ABB RAPID module: Codigo Rappid

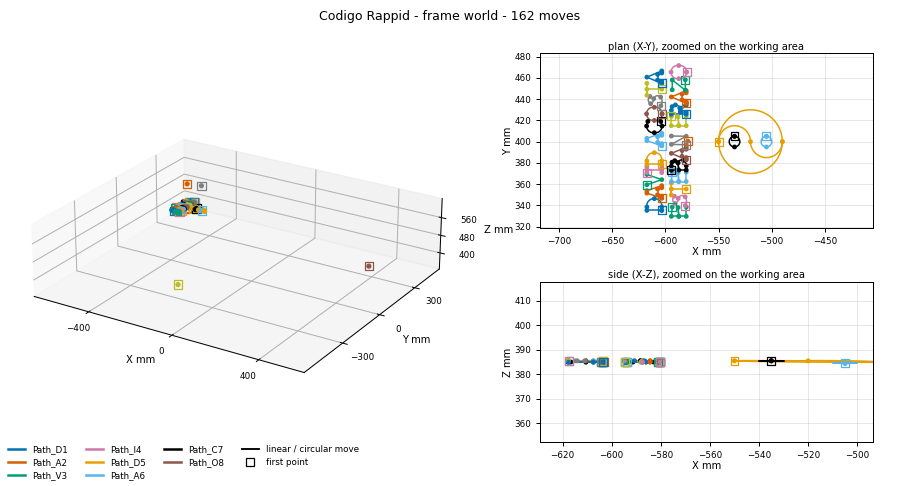
[picture p0: tool path of Codigo Rappid in frame world, 162 of 163 moves have a stored position in this frame; points joined in program order, loops and branches not executed]
MODULE Module1
    PERS tooldata Porta_Marcador:=[TRUE,[[111.723,0,111.723],[0.923879533,0,0.382683432,0]],[1,[0,0,1],[1,0,0,0],0,0,0]];
    TASK PERS wobjdata Workobject_2:=[FALSE,TRUE,"",[[-160,-80,65],[1,0,0,0]],[[-480,560,320],[0,1,0,0]]];
    CONST robtarget Target_10:=[[36.486,144.721,0],[1,0,0,0],[0,0,0,0],[9E+09,9E+09,9E+09,9E+09,9E+09,9E+09]];
    CONST robtarget Target_20:=[[22.486,144.721,-0.5],[1,0,0,0],[0,0,0,0],[9E+09,9E+09,9E+09,9E+09,9E+09,9E+09]];
    CONST robtarget Target_30:=[[22.486,141.533,-0.5],[1,0,0,0],[0,0,0,0],[9E+09,9E+09,9E+09,9E+09,9E+09,9E+09]];
    CONST robtarget Target_40:=[[23.598,136.519,-0.5],[1,0,0,0],[0,0,0,0],[9E+09,9E+09,9E+09,9E+09,9E+09,9E+09]];
    CONST robtarget Target_50:=[[29.498,133.682,0],[1,0,0,0],[0,0,0,0],[9E+09,9E+09,9E+09,9E+09,9E+09,9E+09]];
    CONST robtarget Target_60:=[[35.363,136.541,-0.5],[1,0,0,0],[0,0,0,0],[9E+09,9E+09,9E+09,9E+09,9E+09,9E+09]];
    CONST robtarget Target_70:=[[36.486,141.499,0],[1,0,0,0],[0,0,0,0],[9E+09,9E+09,9E+09,9E+09,9E+09,9E+09]];
    CONST robtarget Target_80:=[[36.486,133.172,-0.5],[1,0,0,0],[0,0,0,0],[9E+09,9E+09,9E+09,9E+09,9E+09,9E+09]];
    CONST robtarget Target_90:=[[22.486,128.452,-0.5],[1,0,0,0],[0,0,0,0],[9E+09,9E+09,9E+09,9E+09,9E+09,9E+09]];
    CONST robtarget Target_100:=[[22.486,126.161,0],[1,0,0,0],[0,0,0,0],[9E+09,9E+09,9E+09,9E+09,9E+09,9E+09]];
    CONST robtarget Target_110:=[[36.486,121.441,-0.5],[1,0,0,0],[0,0,0,0],[9E+09,9E+09,9E+09,9E+09,9E+09,9E+09]];
    CONST robtarget Target_120:=[[36.486,123.404,0],[1,0,0,0],[0,0,0,0],[9E+09,9E+09,9E+09,9E+09,9E+09,9E+09]];
    CONST robtarget Target_130:=[[32.572,124.674,-0.5],[1,0,0,0],[0,0,0,0],[9E+09,9E+09,9E+09,9E+09,9E+09,9E+09]];
    CONST robtarget Target_140:=[[32.572,130.018,0],[1,0,0,0],[0,0,0,0],[9E+09,9E+09,9E+09,9E+09,9E+09,9E+09]];
    CONST robtarget Target_150:=[[36.486,131.289,-0.5],[1,0,0,0],[0,0,0,0],[9E+09,9E+09,9E+09,9E+09,9E+09,9E+09]];
    CONST robtarget Target_160:=[[22.486,120.613,-0.5],[1,0,0,0],[0,0,0,0],[9E+09,9E+09,9E+09,9E+09,9E+09,9E+09]];
    CONST robtarget Target_170:=[[36.486,115.785,-0.5],[1,0,0,0],[0,0,0,0],[9E+09,9E+09,9E+09,9E+09,9E+09,9E+09]];
    CONST robtarget Target_180:=[[22.486,110.907,-0.5],[1,0,0,0],[0,0,0,0],[9E+09,9E+09,9E+09,9E+09,9E+09,9E+09]];
    CONST robtarget Target_190:=[[22.486,109.165,-0.5],[1,0,0,0],[0,0,0,0],[9E+09,9E+09,9E+09,9E+09,9E+09,9E+09]];
    CONST robtarget Target_200:=[[22.486,103.742,-0.5],[1,0,0,0],[0,0,0,0],[9E+09,9E+09,9E+09,9E+09,9E+09,9E+09]];
    CONST robtarget Target_210:=[[22.486,106.454,-0.5],[1,0,0,0],[0,0,0,0],[9E+09,9E+09,9E+09,9E+09,9E+09,9E+09]];
    CONST robtarget Target_220:=[[36.486,106.454,-0.25],[1,0,0,0],[0,0,0,0],[9E+09,9E+09,9E+09,9E+09,9E+09,9E+09]];
    CONST robtarget Target_230:=[[36.486,109.165,-0.25],[1,0,0,0],[0,0,0,0],[9E+09,9E+09,9E+09,9E+09,9E+09,9E+09]];
    CONST robtarget Target_240:=[[36.486,103.742,0],[1,0,0,0],[0,0,0,0],[9E+09,9E+09,9E+09,9E+09,9E+09,9E+09]];
    CONST robtarget Target_250:=[[36.486,101.439,0],[1,0,0,0],[0,0,0,0],[9E+09,9E+09,9E+09,9E+09,9E+09,9E+09]];
    CONST robtarget Target_260:=[[22.486,101.439,-0.5],[1,0,0,0],[0,0,0,0],[9E+09,9E+09,9E+09,9E+09,9E+09,9E+09]];
    CONST robtarget Target_270:=[[22.486,98.251,-0.5],[1,0,0,0],[0,0,0,0],[9E+09,9E+09,9E+09,9E+09,9E+09,9E+09]];
    CONST robtarget Target_280:=[[23.598,93.237,-0.5],[1,0,0,0],[0,0,0,0],[9E+09,9E+09,9E+09,9E+09,9E+09,9E+09]];
    CONST robtarget Target_290:=[[29.498,90.4,0],[1,0,0,0],[0,0,0,0],[9E+09,9E+09,9E+09,9E+09,9E+09,9E+09]];
    CONST robtarget Target_300:=[[35.363,93.259,0],[1,0,0,0],[0,0,0,0],[9E+09,9E+09,9E+09,9E+09,9E+09,9E+09]];
    CONST robtarget Target_310:=[[36.486,98.217,0],[1,0,0,0],[0,0,0,0],[9E+09,9E+09,9E+09,9E+09,9E+09,9E+09]];
    CONST robtarget Target_320:=[[36.486,83.877,0],[1,0,0,0],[0,0,0,0],[9E+09,9E+09,9E+09,9E+09,9E+09,9E+09]];
    CONST robtarget Target_330:=[[22.486,79.157,-0.5],[1,0,0,0],[0,0,0,0],[9E+09,9E+09,9E+09,9E+09,9E+09,9E+09]];
    CONST robtarget Target_340:=[[22.486,76.866,-0.5],[1,0,0,0],[0,0,0,0],[9E+09,9E+09,9E+09,9E+09,9E+09,9E+09]];
    CONST robtarget Target_350:=[[36.486,72.146,0],[1,0,0,0],[0,0,0,0],[9E+09,9E+09,9E+09,9E+09,9E+09,9E+09]];
    CONST robtarget Target_360:=[[36.486,74.109,0],[1,0,0,0],[0,0,0,0],[9E+09,9E+09,9E+09,9E+09,9E+09,9E+09]];
    CONST robtarget Target_370:=[[32.572,75.379,-0.5],[1,0,0,0],[0,0,0,0],[9E+09,9E+09,9E+09,9E+09,9E+09,9E+09]];
    CONST robtarget Target_380:=[[32.572,80.723,0],[1,0,0,0],[0,0,0,0],[9E+09,9E+09,9E+09,9E+09,9E+09,9E+09]];
    CONST robtarget Target_390:=[[36.486,81.994,0],[1,0,0,0],[0,0,0,0],[9E+09,9E+09,9E+09,9E+09,9E+09,9E+09]];
    CONST robtarget Target_400:=[[35.533,60.994,0],[1,0,0,0],[0,0,0,0],[9E+09,9E+09,9E+09,9E+09,9E+09,9E+09]];
    CONST robtarget Target_410:=[[36.328,62.854,0],[1,0,0,0],[0,0,0,0],[9E+09,9E+09,9E+09,9E+09,9E+09,9E+09]];
    CONST robtarget Target_420:=[[36.736,65.35,0],[1,0,0,0],[0,0,0,0],[9E+09,9E+09,9E+09,9E+09,9E+09,9E+09]];
    CONST robtarget Target_430:=[[34.898,69.854,0],[1,0,0,0],[0,0,0,0],[9E+09,9E+09,9E+09,9E+09,9E+09,9E+09]];
    CONST robtarget Target_440:=[[29.498,71.613,0],[1,0,0,0],[0,0,0,0],[9E+09,9E+09,9E+09,9E+09,9E+09,9E+09]];
    CONST robtarget Target_450:=[[24.165,69.866,-0.5],[1,0,0,0],[0,0,0,0],[9E+09,9E+09,9E+09,9E+09,9E+09,9E+09]];
    CONST robtarget Target_460:=[[22.237,65.316,0],[1,0,0,0],[0,0,0,0],[9E+09,9E+09,9E+09,9E+09,9E+09,9E+09]];
    CONST robtarget Target_470:=[[22.6,62.854,0],[1,0,0,0],[0,0,0,0],[9E+09,9E+09,9E+09,9E+09,9E+09,9E+09]];
    CONST robtarget Target_480:=[[23.417,60.994,0],[1,0,0,0],[0,0,0,0],[9E+09,9E+09,9E+09,9E+09,9E+09,9E+09]];
    CONST robtarget Target_490:=[[36.781,53.869,0],[1,0,0,0],[0,0,0,0],[9E+09,9E+09,9E+09,9E+09,9E+09,9E+09]];
    CONST robtarget Target_500:=[[34.875,58.384,0],[1,0,0,0],[0,0,0,0],[9E+09,9E+09,9E+09,9E+09,9E+09,9E+09]];
    CONST robtarget Target_510:=[[29.486,60.052,-0.5],[1,0,0,0],[0,0,0,0],[9E+09,9E+09,9E+09,9E+09,9E+09,9E+09]];
    CONST robtarget Target_520:=[[24.086,58.373,-0.5],[1,0,0,0],[0,0,0,0],[9E+09,9E+09,9E+09,9E+09,9E+09,9E+09]];
    CONST robtarget Target_530:=[[22.191,53.869,-0.5],[1,0,0,0],[0,0,0,0],[9E+09,9E+09,9E+09,9E+09,9E+09,9E+09]];
    CONST robtarget Target_540:=[[24.086,49.353,-0.5],[1,0,0,0],[0,0,0,0],[9E+09,9E+09,9E+09,9E+09,9E+09,9E+09]];
    CONST robtarget Target_550:=[[29.486,47.674,-0.5],[1,0,0,0],[0,0,0,0],[9E+09,9E+09,9E+09,9E+09,9E+09,9E+09]];
    CONST robtarget Target_560:=[[34.875,49.353,-0.5],[1,0,0,0],[0,0,0,0],[9E+09,9E+09,9E+09,9E+09,9E+09,9E+09]];
    CONST robtarget Target_570:=[[35.647,46.324,0],[1,0,0,0],[0,0,0,0],[9E+09,9E+09,9E+09,9E+09,9E+09,9E+09]];
    CONST robtarget Target_580:=[[36.736,41.729,0],[1,0,0,0],[0,0,0,0],[9E+09,9E+09,9E+09,9E+09,9E+09,9E+09]];
    CONST robtarget Target_590:=[[35.465,38.076,0],[1,0,0,0],[0,0,0,0],[9E+09,9E+09,9E+09,9E+09,9E+09,9E+09]];
    CONST robtarget Target_600:=[[32.493,36.806,0],[1,0,0,0],[0,0,0,0],[9E+09,9E+09,9E+09,9E+09,9E+09,9E+09]];
    CONST robtarget Target_610:=[[28.964,39.585,-0.5],[1,0,0,0],[0,0,0,0],[9E+09,9E+09,9E+09,9E+09,9E+09,9E+09]];
    CONST robtarget Target_620:=[[28.227,42.456,-0.5],[1,0,0,0],[0,0,0,0],[9E+09,9E+09,9E+09,9E+09,9E+09,9E+09]];
    CONST robtarget Target_630:=[[26.049,44.282,-0.5],[1,0,0,0],[0,0,0,0],[9E+09,9E+09,9E+09,9E+09,9E+09,9E+09]];
    CONST robtarget Target_640:=[[23.848,41.389,-0.5],[1,0,0,0],[0,0,0,0],[9E+09,9E+09,9E+09,9E+09,9E+09,9E+09]];
    CONST robtarget Target_650:=[[25.368,37.486,-0.5],[1,0,0,0],[0,0,0,0],[9E+09,9E+09,9E+09,9E+09,9E+09,9E+09]];
    CONST robtarget Target_660:=[[36.486,30.713,-0.5],[1,0,0,0],[0,0,0,0],[9E+09,9E+09,9E+09,9E+09,9E+09,9E+09]];
    CONST robtarget Target_670:=[[22.486,30.713,-0.5],[1,0,0,0],[0,0,0,0],[9E+09,9E+09,9E+09,9E+09,9E+09,9E+09]];
    CONST robtarget Target_680:=[[22.486,36.34,-0.5],[1,0,0,0],[0,0,0,0],[9E+09,9E+09,9E+09,9E+09,9E+09,9E+09]];
    CONST robtarget Target_690:=[[22.486,25.086,-0.5],[1,0,0,0],[0,0,0,0],[9E+09,9E+09,9E+09,9E+09,9E+09,9E+09]];
    CONST robtarget Target_770:=[[36.486,25.177,0],[1,0,0,0],[0,0,0,0],[9E+09,9E+09,9E+09,9E+09,9E+09,9E+09]];
    CONST robtarget Target_780:=[[22.486,19.311,0],[1,0,0,0],[0,0,0,0],[9E+09,9E+09,9E+09,9E+09,9E+09,9E+09]];
    CONST robtarget Target_790:=[[36.486,13.446,0],[1,0,0,0],[0,0,0,0],[9E+09,9E+09,9E+09,9E+09,9E+09,9E+09]];
    CONST robtarget Target_800:=[[36.486,15.409,0],[1,0,0,0],[0,0,0,0],[9E+09,9E+09,9E+09,9E+09,9E+09,9E+09]];
    CONST robtarget Target_810:=[[32.572,16.679,0],[1,0,0,0],[0,0,0,0],[9E+09,9E+09,9E+09,9E+09,9E+09,9E+09]];
    CONST robtarget Target_820:=[[32.572,22.023,0],[1,0,0,0],[0,0,0,0],[9E+09,9E+09,9E+09,9E+09,9E+09,9E+09]];
    CONST robtarget Target_830:=[[36.486,23.293,0],[1,0,0,0],[0,0,0,0],[9E+09,9E+09,9E+09,9E+09,9E+09,9E+09]];
    CONST robtarget Target_Pastel_inicio:=[[61.043181897,79.487763711,-109.905526816],[0.928113719,0.029025657,-0.074070087,0.363697757],[1,-1,0,0],[9E+09,9E+09,9E+09,9E+09,9E+09,9E+09]];
    CONST robtarget Target_840:=[[46.365,141.579,0],[1,0,0,0],[0,0,0,0],[9E+09,9E+09,9E+09,9E+09,9E+09,9E+09]];
    CONST robtarget Target_850:=[[45.537,150.337,0],[1,0,0,0],[0,0,0,0],[9E+09,9E+09,9E+09,9E+09,9E+09,9E+09]];
    CONST robtarget Target_860:=[[52.537,150.337,0],[1,0,0,0],[0,0,0,0],[9E+09,9E+09,9E+09,9E+09,9E+09,9E+09]];
    CONST robtarget Target_870:=[[51.856,142.044,0],[1,0,0,0],[0,0,0,0],[9E+09,9E+09,9E+09,9E+09,9E+09,9E+09]];
    CONST robtarget Target_880:=[[59.537,150.337,0],[1,0,0,0],[0,0,0,0],[9E+09,9E+09,9E+09,9E+09,9E+09,9E+09]];
    CONST robtarget Target_890:=[[59.537,141.579,0],[1,0,0,0],[0,0,0,0],[9E+09,9E+09,9E+09,9E+09,9E+09,9E+09]];
    CONST robtarget Target_900:=[[58.697,140.229,0],[1,0,0,0],[0,0,0,0],[9E+09,9E+09,9E+09,9E+09,9E+09,9E+09]];
    CONST robtarget Target_910:=[[59.787,135.634,0],[1,0,0,0],[0,0,0,0],[9E+09,9E+09,9E+09,9E+09,9E+09,9E+09]];
    CONST robtarget Target_920:=[[58.516,131.981,0],[1,0,0,0],[0,0,0,0],[9E+09,9E+09,9E+09,9E+09,9E+09,9E+09]];
    CONST robtarget Target_930:=[[55.543,130.71,0],[1,0,0,0],[0,0,0,0],[9E+09,9E+09,9E+09,9E+09,9E+09,9E+09]];
    CONST robtarget Target_940:=[[52.015,133.49,-0.5],[1,0,0,0],[0,0,0,0],[9E+09,9E+09,9E+09,9E+09,9E+09,9E+09]];
    CONST robtarget Target_950:=[[51.278,136.36,-0.5],[1,0,0,0],[0,0,0,0],[9E+09,9E+09,9E+09,9E+09,9E+09,9E+09]];
    CONST robtarget Target_960:=[[49.099,138.186,-0.5],[1,0,0,0],[0,0,0,0],[9E+09,9E+09,9E+09,9E+09,9E+09,9E+09]];
    CONST robtarget Target_970:=[[46.898,135.293,0],[1,0,0,0],[0,0,0,0],[9E+09,9E+09,9E+09,9E+09,9E+09,9E+09]];
    CONST robtarget Target_980:=[[48.419,131.391,0],[1,0,0,0],[0,0,0,0],[9E+09,9E+09,9E+09,9E+09,9E+09,9E+09]];
    CONST robtarget Target_990:=[[59.537,124.618,0],[1,0,0,0],[0,0,0,0],[9E+09,9E+09,9E+09,9E+09,9E+09,9E+09]];
    CONST robtarget Target_1000:=[[45.537,124.618,-0.5],[1,0,0,0],[0,0,0,0],[9E+09,9E+09,9E+09,9E+09,9E+09,9E+09]];
    CONST robtarget Target_1010:=[[45.537,130.245,-0.5],[1,0,0,0],[0,0,0,0],[9E+09,9E+09,9E+09,9E+09,9E+09,9E+09]];
    CONST robtarget Target_1020:=[[45.537,118.99,0],[1,0,0,0],[0,0,0,0],[9E+09,9E+09,9E+09,9E+09,9E+09,9E+09]];
    CONST robtarget Target_1030:=[[46.365,108.814,0],[1,0,0,0],[0,0,0,0],[9E+09,9E+09,9E+09,9E+09,9E+09,9E+09]];
    CONST robtarget Target_1040:=[[45.537,117.572,-0.5],[1,0,0,0],[0,0,0,0],[9E+09,9E+09,9E+09,9E+09,9E+09,9E+09]];
    CONST robtarget Target_1050:=[[52.537,117.572,-0.5],[1,0,0,0],[0,0,0,0],[9E+09,9E+09,9E+09,9E+09,9E+09,9E+09]];
    CONST robtarget Target_1060:=[[51.856,109.279,-0.5],[1,0,0,0],[0,0,0,0],[9E+09,9E+09,9E+09,9E+09,9E+09,9E+09]];
    CONST robtarget Target_1070:=[[59.537,117.572,-0.5],[1,0,0,0],[0,0,0,0],[9E+09,9E+09,9E+09,9E+09,9E+09,9E+09]];
    CONST robtarget Target_1080:=[[59.537,108.814,0],[1,0,0,0],[0,0,0,0],[9E+09,9E+09,9E+09,9E+09,9E+09,9E+09]];
    CONST robtarget Target_1090:=[[45.537,106.772,0],[1,0,0,0],[0,0,0,0],[9E+09,9E+09,9E+09,9E+09,9E+09,9E+09]];
    CONST robtarget Target_1100:=[[59.537,106.772,0],[1,0,0,0],[0,0,0,0],[9E+09,9E+09,9E+09,9E+09,9E+09,9E+09]];
    CONST robtarget Target_1110:=[[59.537,102.755,0],[1,0,0,0],[0,0,0,0],[9E+09,9E+09,9E+09,9E+09,9E+09,9E+09]];
    CONST robtarget Target_1120:=[[59.276,100.424,0],[1,0,0,0],[0,0,0,0],[9E+09,9E+09,9E+09,9E+09,9E+09,9E+09]];
    CONST robtarget Target_1130:=[[57.081,97.673,0],[1,0,0,0],[0,0,0,0],[9E+09,9E+09,9E+09,9E+09,9E+09,9E+09]];
    CONST robtarget Target_1140:=[[52.996,97.962,0],[1,0,0,0],[0,0,0,0],[9E+09,9E+09,9E+09,9E+09,9E+09,9E+09]];
    CONST robtarget Target_1150:=[[51.754,99.896,-0.5],[1,0,0,0],[0,0,0,0],[9E+09,9E+09,9E+09,9E+09,9E+09,9E+09]];
    CONST robtarget Target_1160:=[[52.537,106.772,-0.5],[1,0,0,0],[0,0,0,0],[9E+09,9E+09,9E+09,9E+09,9E+09,9E+09]];
    CONST robtarget Target_1170:=[[50.461,98.456,0],[1,0,0,0],[0,0,0,0],[9E+09,9E+09,9E+09,9E+09,9E+09,9E+09]];
    CONST robtarget Target_1180:=[[48.691,97.934,0],[1,0,0,0],[0,0,0,0],[9E+09,9E+09,9E+09,9E+09,9E+09,9E+09]];
    CONST robtarget Target_1190:=[[47.154,98.28,0],[1,0,0,0],[0,0,0,0],[9E+09,9E+09,9E+09,9E+09,9E+09,9E+09]];
    CONST robtarget Target_1200:=[[46.104,99.386,0],[1,0,0,0],[0,0,0,0],[9E+09,9E+09,9E+09,9E+09,9E+09,9E+09]];
    CONST robtarget Target_1210:=[[45.537,103.062,-0.5],[1,0,0,0],[0,0,0,0],[9E+09,9E+09,9E+09,9E+09,9E+09,9E+09]];
    CONST robtarget Target_1220:=[[59.537,96.935,0],[1,0,0,0],[0,0,0,0],[9E+09,9E+09,9E+09,9E+09,9E+09,9E+09]];
    CONST robtarget Target_1230:=[[45.537,91.07,-0.5],[1,0,0,0],[0,0,0,0],[9E+09,9E+09,9E+09,9E+09,9E+09,9E+09]];
    CONST robtarget Target_1240:=[[59.537,85.204,0],[1,0,0,0],[0,0,0,0],[9E+09,9E+09,9E+09,9E+09,9E+09,9E+09]];
    CONST robtarget Target_1250:=[[59.537,87.167,0],[1,0,0,0],[0,0,0,0],[9E+09,9E+09,9E+09,9E+09,9E+09,9E+09]];
    CONST robtarget Target_1260:=[[55.623,88.438,-0.5],[1,0,0,0],[0,0,0,0],[9E+09,9E+09,9E+09,9E+09,9E+09,9E+09]];
    CONST robtarget Target_1270:=[[55.623,93.781,0],[1,0,0,0],[0,0,0,0],[9E+09,9E+09,9E+09,9E+09,9E+09,9E+09]];
    CONST robtarget Target_1280:=[[59.537,95.052,0],[1,0,0,0],[0,0,0,0],[9E+09,9E+09,9E+09,9E+09,9E+09,9E+09]];
    CONST robtarget Target_1290:=[[59.537,83.009,0],[1,0,0,0],[0,0,0,0],[9E+09,9E+09,9E+09,9E+09,9E+09,9E+09]];
    CONST robtarget Target_1300:=[[45.537,82.555,-0.5],[1,0,0,0],[0,0,0,0],[9E+09,9E+09,9E+09,9E+09,9E+09,9E+09]];
    CONST robtarget Target_1310:=[[59.537,74.903,0],[1,0,0,0],[0,0,0,0],[9E+09,9E+09,9E+09,9E+09,9E+09,9E+09]];
    CONST robtarget Target_1320:=[[45.537,74.727,-0.5],[1,0,0,0],[0,0,0,0],[9E+09,9E+09,9E+09,9E+09,9E+09,9E+09]];
    CONST robtarget Target_1340:=[[45.537,56.251,0],[1,0,0,0],[0,0,0,0],[9E+09,9E+09,9E+09,9E+09,9E+09,9E+09]];
    CONST robtarget Target_1350:=[[45.537,65.01,-0.5],[1,0,0,0],[0,0,0,0],[9E+09,9E+09,9E+09,9E+09,9E+09,9E+09]];
    CONST robtarget Target_1360:=[[52.537,65.01,-0.5],[1,0,0,0],[0,0,0,0],[9E+09,9E+09,9E+09,9E+09,9E+09,9E+09]];
    CONST robtarget Target_1370:=[[51.856,56.716,0],[1,0,0,0],[0,0,0,0],[9E+09,9E+09,9E+09,9E+09,9E+09,9E+09]];
    CONST robtarget Target_1380:=[[59.537,65.01,0],[1,0,0,0],[0,0,0,0],[9E+09,9E+09,9E+09,9E+09,9E+09,9E+09]];
    CONST robtarget Target_1390:=[[59.537,56.251,0],[1,0,0,0],[0,0,0,0],[9E+09,9E+09,9E+09,9E+09,9E+09,9E+09]];
    CONST robtarget Target_1400:=[[59.537,54.209,0],[1,0,0,0],[0,0,0,0],[9E+09,9E+09,9E+09,9E+09,9E+09,9E+09]];
    CONST robtarget Target_1410:=[[45.537,54.209,0],[1,0,0,0],[0,0,0,0],[9E+09,9E+09,9E+09,9E+09,9E+09,9E+09]];
    CONST robtarget Target_1420:=[[45.537,50.601,-0.5],[1,0,0,0],[0,0,0,0],[9E+09,9E+09,9E+09,9E+09,9E+09,9E+09]];
    CONST robtarget Target_1430:=[[45.667,48.588,-0.5],[1,0,0,0],[0,0,0,0],[9E+09,9E+09,9E+09,9E+09,9E+09,9E+09]];
    CONST robtarget Target_1440:=[[46.274,47.039,-0.5],[1,0,0,0],[0,0,0,0],[9E+09,9E+09,9E+09,9E+09,9E+09,9E+09]];
    CONST robtarget Target_1450:=[[47.494,45.876,-0.5],[1,0,0,0],[0,0,0,0],[9E+09,9E+09,9E+09,9E+09,9E+09,9E+09]];
    CONST robtarget Target_1460:=[[49.338,45.451,-0.5],[1,0,0,0],[0,0,0,0],[9E+09,9E+09,9E+09,9E+09,9E+09,9E+09]];
    CONST robtarget Target_1470:=[[51.907,46.233,-0.5],[1,0,0,0],[0,0,0,0],[9E+09,9E+09,9E+09,9E+09,9E+09,9E+09]];
    CONST robtarget Target_1480:=[[53.445,48.355,-0.5],[1,0,0,0],[0,0,0,0],[9E+09,9E+09,9E+09,9E+09,9E+09,9E+09]];
    CONST robtarget Target_1490:=[[59.537,43.84,0],[1,0,0,0],[0,0,0,0],[9E+09,9E+09,9E+09,9E+09,9E+09,9E+09]];
    CONST robtarget Target_1500:=[[59.537,45.791,0],[1,0,0,0],[0,0,0,0],[9E+09,9E+09,9E+09,9E+09,9E+09,9E+09]];
    CONST robtarget Target_1510:=[[53.966,50.216,0],[1,0,0,0],[0,0,0,0],[9E+09,9E+09,9E+09,9E+09,9E+09,9E+09]];
    CONST robtarget Target_1520:=[[53.966,52.349,0],[1,0,0,0],[0,0,0,0],[9E+09,9E+09,9E+09,9E+09,9E+09,9E+09]];
    CONST robtarget Target_1530:=[[59.537,52.349,0],[1,0,0,0],[0,0,0,0],[9E+09,9E+09,9E+09,9E+09,9E+09,9E+09]];
    CONST robtarget Target_1540:=[[59.537,43.84,0],[1,0,0,0],[0,0,0,0],[9E+09,9E+09,9E+09,9E+09,9E+09,9E+09]];
    CONST robtarget Target_1550:=[[45.537,37.906,-0.5],[1,0,0,0],[0,0,0,0],[9E+09,9E+09,9E+09,9E+09,9E+09,9E+09]];
    CONST robtarget Target_1560:=[[59.537,32.041,0],[1,0,0,0],[0,0,0,0],[9E+09,9E+09,9E+09,9E+09,9E+09,9E+09]];
    CONST robtarget Target_1570:=[[59.537,34.003,-0.25],[1,0,0,0],[0,0,0,0],[9E+09,9E+09,9E+09,9E+09,9E+09,9E+09]];
    CONST robtarget Target_1580:=[[55.623,35.274,-0.5],[1,0,0,0],[0,0,0,0],[9E+09,9E+09,9E+09,9E+09,9E+09,9E+09]];
    CONST robtarget Target_1590:=[[55.623,40.618,0],[1,0,0,0],[0,0,0,0],[9E+09,9E+09,9E+09,9E+09,9E+09,9E+09]];
    CONST robtarget Target_1600:=[[59.537,41.888,-0.25],[1,0,0,0],[0,0,0,0],[9E+09,9E+09,9E+09,9E+09,9E+09,9E+09]];
    CONST robtarget Target_1610:=[[58.709,21.785,0],[1,0,0,0],[0,0,0,0],[9E+09,9E+09,9E+09,9E+09,9E+09,9E+09]];
    CONST robtarget Target_1620:=[[58.669,31.564,-0.5],[1,0,0,0],[0,0,0,0],[9E+09,9E+09,9E+09,9E+09,9E+09,9E+09]];
    CONST robtarget Target_1630:=[[46.377,21.977,0],[1,0,0,0],[0,0,0,0],[9E+09,9E+09,9E+09,9E+09,9E+09,9E+09]];
    CONST robtarget Target_1640:=[[46.365,31.224,-0.5],[1,0,0,0],[0,0,0,0],[9E+09,9E+09,9E+09,9E+09,9E+09,9E+09]];
    CONST robtarget Target_1650:=[[59.832,14.558,0],[1,0,0,0],[0,0,0,0],[9E+09,9E+09,9E+09,9E+09,9E+09,9E+09]];
    CONST robtarget Target_1660:=[[57.926,19.073,0],[1,0,0,0],[0,0,0,0],[9E+09,9E+09,9E+09,9E+09,9E+09,9E+09]];
    CONST robtarget Target_1670:=[[52.537,20.741,0],[1,0,0,0],[0,0,0,0],[9E+09,9E+09,9E+09,9E+09,9E+09,9E+09]];
    CONST robtarget Target_1680:=[[47.137,19.062,-0.5],[1,0,0,0],[0,0,0,0],[9E+09,9E+09,9E+09,9E+09,9E+09,9E+09]];
    CONST robtarget Target_1690:=[[45.242,14.558,-0.5],[1,0,0,0],[0,0,0,0],[9E+09,9E+09,9E+09,9E+09,9E+09,9E+09]];
    CONST robtarget Target_1700:=[[47.137,10.042,-0.5],[1,0,0,0],[0,0,0,0],[9E+09,9E+09,9E+09,9E+09,9E+09,9E+09]];
    CONST robtarget Target_1710:=[[52.537,8.363,0],[1,0,0,0],[0,0,0,0],[9E+09,9E+09,9E+09,9E+09,9E+09,9E+09]];
    CONST robtarget Target_1720:=[[57.926,10.042,0],[1,0,0,0],[0,0,0,0],[9E+09,9E+09,9E+09,9E+09,9E+09,9E+09]];
    CONST robtarget Target_1880:=[[90,80,-0.5],[1,0,0,0],[1,0,-1,0],[9E+09,9E+09,9E+09,9E+09,9E+09,9E+09]];
    CONST robtarget Target_1890:=[[120,110,-0.5],[1,0,0,0],[1,0,-1,0],[9E+09,9E+09,9E+09,9E+09,9E+09,9E+09]];
    CONST robtarget Target_1900:=[[150,80,0],[1,0,0,0],[1,0,-1,0],[9E+09,9E+09,9E+09,9E+09,9E+09,9E+09]];
    CONST robtarget Target_1910:=[[120,50,0],[1,0,0,0],[1,0,-1,0],[9E+09,9E+09,9E+09,9E+09,9E+09,9E+09]];
    CONST robtarget Target_1920:=[[105,65,-0.5],[1,0,0,0],[1,0,-1,0],[9E+09,9E+09,9E+09,9E+09,9E+09,9E+09]];
    CONST robtarget Target_1930:=[[120,80,-0.5],[1,0,0,0],[1,0,-1,0],[9E+09,9E+09,9E+09,9E+09,9E+09,9E+09]];
    CONST robtarget Target_1940:=[[135,95,-0.5],[1,0,0,0],[0,0,0,0],[9E+09,9E+09,9E+09,9E+09,9E+09,9E+09]];
    CONST robtarget Target_1800:=[[135,75,0.5],[1,0,0,0],[0,0,0,0],[9E+09,9E+09,9E+09,9E+09,9E+09,9E+09]];
    CONST robtarget Target_1810:=[[139.999,79.929,0.5],[1,0,0,0],[0,0,0,0],[9E+09,9E+09,9E+09,9E+09,9E+09,9E+09]];
    CONST robtarget Target_1820:=[[135.031,85,0.5],[1,0,0,0],[0,0,0,0],[9E+09,9E+09,9E+09,9E+09,9E+09,9E+09]];
    CONST robtarget Target_1830:=[[130,79.971,0.5],[1,0,0,0],[0,0,0,0],[9E+09,9E+09,9E+09,9E+09,9E+09,9E+09]];
    CONST robtarget Target_1840:=[[104.983,75,-0.5],[1,0,0,0],[0,0,0,0],[9E+09,9E+09,9E+09,9E+09,9E+09,9E+09]];
    CONST robtarget Target_1850:=[[110,80.057,-0.5],[1,0,0,0],[0,0,0,0],[9E+09,9E+09,9E+09,9E+09,9E+09,9E+09]];
    CONST robtarget Target_1860:=[[105.013,85,-0.5],[1,0,0,0],[0,0,0,0],[9E+09,9E+09,9E+09,9E+09,9E+09,9E+09]];
    CONST robtarget Target_1870:=[[100.001,79.927,-0.5],[1,0,0,0],[0,0,0,0],[9E+09,9E+09,9E+09,9E+09,9E+09,9E+09]];
    CONST robtarget HOME:=[[1187.185107433,480,-141.883543813],[0,0.130526193,0,0.991444861],[0,0,0,0],[9E+09,9E+09,9E+09,9E+09,9E+09,9E+09]];
    CONST robtarget Target_No_Golpear:=[[248.163091014,252.745660701,-202.50817905],[0.921868667,0.051152682,-0.130535664,0.361250611],[1,-1,0,0],[9E+09,9E+09,9E+09,9E+09,9E+09,9E+09]];
    CONST jointtarget HOME_IR:=[[0,0,0,0,0,0],[9E+09,9E+09,9E+09,9E+09,9E+09,9E+09]];
    CONST robtarget Target_Mantenimiento:=[[640,1027.185107433,-141.883543813],[0.701057385,-0.092295956,-0.092295956,-0.701057385],[-2,-1,0,0],[9E+09,9E+09,9E+09,9E+09,9E+09,9E+09]];

    PROC main()

        WHILE TRUE DO
            Reset DO_01;
            Reset DO_02;
            Reset Conveyor_FWD;
            Reset Conveyor_INV;
            IF DI_01 = 1 AND DI_02=0 THEN
            Set Conveyor_FWD;
            Set DO_01;
            WaitTime 4;
            Reset Conveyor_FWD;
                Path_No_Golpear;
                Path_Pastel_Inicio;
                Path_D1;
                Path_Pastel_Inicio;
                Path_A2;
                Path_Pastel_Inicio;
                Path_V3;
                Path_Pastel_Inicio;
                Path_I4;
                Path_Pastel_Inicio;
                Path_D5;
                Path_Pastel_Inicio;
                Path_A6;
                Path_Pastel_Inicio;
                Path_C7;
                Path_Pastel_Inicio;
                Path_O8;
                Path_Pastel_Inicio;
                Path_S9;
                Path_Pastel_Inicio;
                Path_T10;
                Path_Pastel_Inicio;
                Path_A11;
                Path_Pastel_Inicio;
                Path_1E;
                Path_Pastel_Inicio;
                Path_2S;
                Path_Pastel_Inicio;
                Path_3T;
                Path_Pastel_Inicio;
                Path_4E;
                Path_Pastel_Inicio;
                Path_5B;
                Path_Pastel_Inicio;
                Path_6A;
                Path_Pastel_Inicio;
                Path_7N;
                Path_Pastel_Inicio;
                Path_8E;
                Path_Pastel_Inicio;
                Path_9R;
                Path_Pastel_Inicio;
                Path_10A;
                Path_Pastel_Inicio;
                Path_11Z;
                Path_Pastel_Inicio;
                Path_12O;
                Path_Pastel_Inicio;
                Path_JIM1;
                Path_Pastel_Inicio;
                Path_JAM1;
                Path_Pastel_Inicio;
                Path_JAM2;

                Path_No_Golpear;
                Path_HOME;
                Path_HOME_IR;
                Reset DO_01;
                Reset DO_02;
                Reset Conveyor_FWD;
                Reset Conveyor_INV;

            ELSEIF DI_01 = 0 AND DI_02=1 THEN
                Path_HOME;
                Path_Mantenimiento;
                WaitUntil DI_01=1 AND DI_02=1;

        ENDIF
     ENDWHILE
    ENDPROC


    PROC Path_D1()
        MoveJ Target_10,v100,z1,Porta_Marcador\WObj:=Workobject_2;
        MoveL Target_20,v100,z1,Porta_Marcador\WObj:=Workobject_2;
        MoveL Target_30,v100,z1,Porta_Marcador\WObj:=Workobject_2;
        MoveC Target_40,Target_50,v100,z1,Porta_Marcador\WObj:=Workobject_2;
        MoveC Target_60,Target_70,v100,z1,Porta_Marcador\WObj:=Workobject_2;
        MoveL Target_10,v100,z1,Porta_Marcador\WObj:=Workobject_2;
    ENDPROC
    PROC Path_A2()
        MoveJ Target_80,v100,z1,Porta_Marcador\WObj:=Workobject_2;
        MoveL Target_90,v100,z1,Porta_Marcador\WObj:=Workobject_2;
        MoveL Target_100,v100,z1,Porta_Marcador\WObj:=Workobject_2;
        MoveL Target_110,v100,z1,Porta_Marcador\WObj:=Workobject_2;
        MoveL Target_120,v100,z1,Porta_Marcador\WObj:=Workobject_2;
        MoveL Target_130,v100,z1,Porta_Marcador\WObj:=Workobject_2;
        MoveL Target_140,v100,z1,Porta_Marcador\WObj:=Workobject_2;
        MoveL Target_150,v100,z1,Porta_Marcador\WObj:=Workobject_2;
        MoveL Target_80,v100,z1,Porta_Marcador\WObj:=Workobject_2;
    ENDPROC
    PROC Path_V3()
        MoveJ Target_160,v100,z1,Porta_Marcador\WObj:=Workobject_2;
        MoveL Target_170,v100,z1,Porta_Marcador\WObj:=Workobject_2;
        MoveL Target_180,v100,z1,Porta_Marcador\WObj:=Workobject_2;
    ENDPROC
    PROC Path_I4()
        MoveJ Target_190,v100,z1,Porta_Marcador\WObj:=Workobject_2;
        MoveL Target_200,v100,z1,Porta_Marcador\WObj:=Workobject_2;
        MoveL Target_210,v100,z1,Porta_Marcador\WObj:=Workobject_2;
        MoveL Target_220,v100,z1,Porta_Marcador\WObj:=Workobject_2;
        MoveL Target_230,v100,z1,Porta_Marcador\WObj:=Workobject_2;
        MoveL Target_240,v100,z1,Porta_Marcador\WObj:=Workobject_2;
    ENDPROC
    PROC Path_D5()
        MoveJ Target_250,v100,z1,Porta_Marcador\WObj:=Workobject_2;
        MoveL Target_260,v100,z1,Porta_Marcador\WObj:=Workobject_2;
        MoveL Target_270,v100,z1,Porta_Marcador\WObj:=Workobject_2;
        MoveC Target_280,Target_290,v100,z1,Porta_Marcador\WObj:=Workobject_2;
        MoveC Target_300,Target_310,v100,z1,Porta_Marcador\WObj:=Workobject_2;
        MoveL Target_250,v100,z1,Porta_Marcador\WObj:=Workobject_2;
    ENDPROC
    PROC Path_A6()
        MoveJ Target_320,v100,z1,Porta_Marcador\WObj:=Workobject_2;
        MoveL Target_330,v100,z1,Porta_Marcador\WObj:=Workobject_2;
        MoveL Target_340,v100,z1,Porta_Marcador\WObj:=Workobject_2;
        MoveL Target_350,v100,z1,Porta_Marcador\WObj:=Workobject_2;
        MoveL Target_360,v100,z1,Porta_Marcador\WObj:=Workobject_2;
        MoveL Target_370,v100,z1,Porta_Marcador\WObj:=Workobject_2;
        MoveL Target_380,v100,z1,Porta_Marcador\WObj:=Workobject_2;
        MoveL Target_390,v100,z1,Porta_Marcador\WObj:=Workobject_2;
        MoveL Target_320,v100,z1,Porta_Marcador\WObj:=Workobject_2;
    ENDPROC
    PROC Path_C7()
        MoveJ Target_400,v100,z1,Porta_Marcador\WObj:=Workobject_2;
        MoveC Target_410,Target_420,v100,z1,Porta_Marcador\WObj:=Workobject_2;
        MoveC Target_430,Target_440,v100,z1,Porta_Marcador\WObj:=Workobject_2;
        MoveC Target_450,Target_460,v100,z1,Porta_Marcador\WObj:=Workobject_2;
        MoveC Target_470,Target_480,v100,z1,Porta_Marcador\WObj:=Workobject_2;
    ENDPROC
    PROC Path_O8()
        MoveJ Target_490,v100,z1,Porta_Marcador\WObj:=Workobject_2;
        MoveC Target_500,Target_510,v100,z1,Porta_Marcador\WObj:=Workobject_2;
        MoveC Target_520,Target_530,v100,z1,Porta_Marcador\WObj:=Workobject_2;
        MoveC Target_540,Target_550,v100,z1,Porta_Marcador\WObj:=Workobject_2;
        MoveC Target_560,Target_490,v100,z1,Porta_Marcador\WObj:=Workobject_2;
    ENDPROC
    PROC Path_S9()
        MoveJ Target_570,v100,z1,Porta_Marcador\WObj:=Workobject_2;
        MoveC Target_580,Target_590,v100,z1,Porta_Marcador\WObj:=Workobject_2;
        MoveC Target_600,Target_610,v100,z1,Porta_Marcador\WObj:=Workobject_2;
        MoveC Target_620,Target_630,v100,z1,Porta_Marcador\WObj:=Workobject_2;
        MoveC Target_640,Target_650,v100,z1,Porta_Marcador\WObj:=Workobject_2;
    ENDPROC
    PROC Path_T10()
        MoveJ Target_660,v100,z1,Porta_Marcador\WObj:=Workobject_2;
        MoveL Target_670,v100,z1,Porta_Marcador\WObj:=Workobject_2;
        MoveL Target_680,v100,z1,Porta_Marcador\WObj:=Workobject_2;
        MoveL Target_690,v100,z1,Porta_Marcador\WObj:=Workobject_2;
    ENDPROC
    PROC Path_A11()
        MoveJ Target_770,v100,z1,Porta_Marcador\WObj:=Workobject_2;
        MoveL Target_780,v100,z1,Porta_Marcador\WObj:=Workobject_2;
        MoveL Target_790,v100,z1,Porta_Marcador\WObj:=Workobject_2;
        MoveL Target_800,v100,z1,Porta_Marcador\WObj:=Workobject_2;
        MoveL Target_810,v100,z1,Porta_Marcador\WObj:=Workobject_2;
        MoveL Target_820,v100,z1,Porta_Marcador\WObj:=Workobject_2;
        MoveL Target_830,v100,z1,Porta_Marcador\WObj:=Workobject_2;
        MoveL Target_770,v100,z1,Porta_Marcador\WObj:=Workobject_2;
    ENDPROC
    PROC Path_Pastel_inicio()
        MoveJ Target_Pastel_inicio,v100,z1,Porta_Marcador\WObj:=Workobject_2;
    ENDPROC
    PROC Path_1E()
        MoveJ Target_840,v100,z1,Porta_Marcador\WObj:=Workobject_2;
        MoveL Target_850,v100,z1,Porta_Marcador\WObj:=Workobject_2;
        MoveL Target_860,v100,z1,Porta_Marcador\WObj:=Workobject_2;
        MoveL Target_870,v100,z1,Porta_Marcador\WObj:=Workobject_2;
        MoveL Target_860,v100,z1,Porta_Marcador\WObj:=Workobject_2;
        MoveL Target_880,v100,z1,Porta_Marcador\WObj:=Workobject_2;
        MoveL Target_890,v100,z1,Porta_Marcador\WObj:=Workobject_2;
    ENDPROC
    PROC Path_2S()
        MoveJ Target_900,v100,z1,Porta_Marcador\WObj:=Workobject_2;
        MoveC Target_910,TArget_920,v100,z1,Porta_Marcador\WObj:=Workobject_2;
        MoveC Target_930,Target_940,v100,z1,Porta_Marcador\WObj:=Workobject_2;
        MoveC Target_950,Target_960,v100,z1,Porta_Marcador\WObj:=Workobject_2;
        MoveC Target_970,Target_980,v100,z1,Porta_Marcador\WObj:=Workobject_2;
    ENDPROC
    PROC Path_3T()
        MoveJ Target_990,v100,z1,Porta_Marcador\WObj:=Workobject_2;
        MoveL Target_1000,v100,z1,Porta_Marcador\WObj:=Workobject_2;
        MoveL Target_1010,v100,z1,Porta_Marcador\WObj:=Workobject_2;
        MoveL Target_1020,v100,z1,Porta_Marcador\WObj:=Workobject_2;
    ENDPROC
    PROC Path_4E()
        MoveJ Target_1030,v100,z1,Porta_Marcador\WObj:=Workobject_2;
        MoveL Target_1040,v100,z1,Porta_Marcador\WObj:=Workobject_2;
        MoveL Target_1050,v100,z1,Porta_Marcador\WObj:=Workobject_2;
        MoveL Target_1060,v100,z1,Porta_Marcador\WObj:=Workobject_2;
        MoveL Target_1050,v100,z1,Porta_Marcador\WObj:=Workobject_2;
        MoveL Target_1070,v100,z1,Porta_Marcador\WObj:=Workobject_2;
        MoveL Target_1080,v100,z1,Porta_Marcador\WObj:=Workobject_2;
    ENDPROC
    PROC Path_5B()
        MoveJ Target_1090,v100,z1,Porta_Marcador\WObj:=Workobject_2;
        MoveL Target_1100,v100,z1,Porta_Marcador\WObj:=Workobject_2;
        MoveL Target_1110,v100,z1,Porta_Marcador\WObj:=Workobject_2;
        MoveC Target_1120,Target_1130,v100,z1,Porta_Marcador\WObj:=Workobject_2;
        MoveC Target_1140,Target_1150,v100,z1,Porta_Marcador\WObj:=Workobject_2;
        MoveL Target_1160,v100,z1,Porta_Marcador\WObj:=Workobject_2;
        MoveL Target_1150,v100,z1,Porta_Marcador\WObj:=Workobject_2;
        MoveC Target_1170,Target_1180,v100,z1,Porta_Marcador\WObj:=Workobject_2;
        MoveC Target_1190,Target_1200,v100,z1,Porta_Marcador\WObj:=Workobject_2;
        MoveL Target_1210,v100,z1,Porta_Marcador\WObj:=Workobject_2;
        MoveL Target_1090,v100,z1,Porta_Marcador\WObj:=Workobject_2;
    ENDPROC
    PROC Path_6A()
        MoveJ Target_1220,v100,z1,Porta_Marcador\WObj:=Workobject_2;
        MoveL Target_1230,v100,z1,Porta_Marcador\WObj:=Workobject_2;
        MoveL Target_1240,v100,z1,Porta_Marcador\WObj:=Workobject_2;
        MoveL Target_1250,v100,z1,Porta_Marcador\WObj:=Workobject_2;
        MoveL Target_1260,v100,z1,Porta_Marcador\WObj:=Workobject_2;
        MoveL Target_1270,v100,z1,Porta_Marcador\WObj:=Workobject_2;
        MoveL Target_1280,v100,z1,Porta_Marcador\WObj:=Workobject_2;
        MoveL Target_1220,v100,z1,Porta_Marcador\WObj:=Workobject_2;
    ENDPROC
    PROC Path_7N()
        MoveJ Target_1290,v100,z1,Porta_Marcador\WObj:=Workobject_2;
        MoveL Target_1300,v100,z1,Porta_Marcador\WObj:=Workobject_2;
        MoveL Target_1310,v100,z1,Porta_Marcador\WObj:=Workobject_2;
        MoveL Target_1320,v100,z1,Porta_Marcador\WObj:=Workobject_2;
    ENDPROC
    PROC Path_8E()
        MoveJ Target_1340,v100,z1,Porta_Marcador\WObj:=Workobject_2;
        MoveL Target_1350,v100,z1,Porta_Marcador\WObj:=Workobject_2;
        MoveL Target_1360,v100,z1,Porta_Marcador\WObj:=Workobject_2;
        MoveL Target_1370,v100,z1,Porta_Marcador\WObj:=Workobject_2;
        MoveL Target_1360,v100,z1,Porta_Marcador\WObj:=Workobject_2;
        MoveL Target_1380,v100,z1,Porta_Marcador\WObj:=Workobject_2;
        MoveL Target_1390,v100,z1,Porta_Marcador\WObj:=Workobject_2;
    ENDPROC
    PROC Path_9R()
        MoveJ Target_1400,v100,z1,Porta_Marcador\WObj:=Workobject_2;
        MoveL Target_1410,v100,z1,Porta_Marcador\WObj:=Workobject_2;
        MoveL Target_1420,v100,z1,Porta_Marcador\WObj:=Workobject_2;
        MoveC Target_1430,Target_1440,v100,z1,Porta_Marcador\WObj:=Workobject_2;
        MoveC Target_1450,Target_1460,v100,z1,Porta_Marcador\WObj:=Workobject_2;
        MoveC Target_1470,Target_1480,v100,z1,Porta_Marcador\WObj:=Workobject_2;
        MoveL Target_1490,v100,z1,Porta_Marcador\WObj:=Workobject_2;
        MoveL Target_1500,v100,z1,Porta_Marcador\WObj:=Workobject_2;
        MoveL Target_1510,v100,z1,Porta_Marcador\WObj:=Workobject_2;
        MoveL Target_1520,v100,z1,Porta_Marcador\WObj:=Workobject_2;
        MoveL Target_1530,v100,z1,Porta_Marcador\WObj:=Workobject_2;
    ENDPROC
    PROC Path_10A()
        MoveJ Target_1540,v100,z1,Porta_Marcador\WObj:=Workobject_2;
        MoveL Target_1550,v100,z1,Porta_Marcador\WObj:=Workobject_2;
        MoveL Target_1560,v100,z1,Porta_Marcador\WObj:=Workobject_2;
        MoveL Target_1570,v100,z1,Porta_Marcador\WObj:=Workobject_2;
        MoveL Target_1580,v100,z1,Porta_Marcador\WObj:=Workobject_2;
        MoveL Target_1590,v100,z1,Porta_Marcador\WObj:=Workobject_2;
        MoveL Target_1600,v100,z1,Porta_Marcador\WObj:=Workobject_2;
        MoveL Target_1540,v100,z1,Porta_Marcador\WObj:=Workobject_2;
    ENDPROC
    PROC Path_11Z()
        MoveJ Target_1610,v100,z1,Porta_Marcador\WObj:=Workobject_2;
        MoveL Target_1620,v100,z1,Porta_Marcador\WObj:=Workobject_2;
        MoveL Target_1630,v100,z1,Porta_Marcador\WObj:=Workobject_2;
        MoveL Target_1640,v100,z1,Porta_Marcador\WObj:=Workobject_2;
    ENDPROC
    PROC Path_12O()
        MoveJ Target_1650,v100,z1,Porta_Marcador\WObj:=Workobject_2;
        MoveC Target_1660,Target_1670,v100,z1,Porta_Marcador\WObj:=Workobject_2;
        MoveC Target_1680,Target_1690,v100,z1,Porta_Marcador\WObj:=Workobject_2;
        MoveC Target_1700,Target_1710,v100,z1,Porta_Marcador\WObj:=Workobject_2;
        MoveC Target_1720,Target_1650,v100,z1,Porta_Marcador\WObj:=Workobject_2;
    ENDPROC
    PROC Path_JIM1()
        MoveJ Target_1880,v100,z1,Porta_Marcador\WObj:=Workobject_2;
        MoveC Target_1890,Target_1900,v100,z1,Porta_Marcador\WObj:=Workobject_2;
        MoveC Target_1910,Target_1880,v100,z1,Porta_Marcador\WObj:=Workobject_2;
        MoveC Target_1920,Target_1930,v100,z1,Porta_Marcador\WObj:=Workobject_2;
        MoveC Target_1940,Target_1900,v100,z1,Porta_Marcador\WObj:=Workobject_2;
    ENDPROC
    PROC Path_JAM1()
        MoveJ Target_1800,v100,z1,Porta_Marcador\WObj:=Workobject_2;
        MoveC Target_1810,Target_1820,v100,z1,Porta_Marcador\WObj:=Workobject_2;
        MoveC Target_1830,Target_1800,v100,z1,Porta_Marcador\WObj:=Workobject_2;
    ENDPROC
    PROC Path_JAM2()
        MoveJ Target_1840,v100,z1,Porta_Marcador\WObj:=Workobject_2;
        MoveC Target_1850,Target_1860,v100,z1,Porta_Marcador\WObj:=Workobject_2;
        MoveC Target_1870,Target_1840,v100,z1,Porta_Marcador\WObj:=Workobject_2;
    ENDPROC
    PROC Path_HOME()
        MoveJ HOME,v1000,z100,Porta_Marcador\WObj:=Workobject_2;
    ENDPROC
    PROC Path_No_Golpear()
        MoveJ Target_No_Golpear,v100,z1,Porta_Marcador\WObj:=Workobject_2;
    ENDPROC
    PROC Path_Mantenimiento()
        MoveL Target_Mantenimiento,v1000,z100,Porta_Marcador\WObj:=Workobject_2;
    ENDPROC
    PROC Path_HOME_IR()
        MoveAbsJ HOME_IR,V300,fine,Porta_Marcador;
    ENDPROC
ENDMODULE
